TYPE "UDT_Recipe"
STRUCT
    name     : String[16];
    tempSet  : Real;
    mixTime  : Time;
END_STRUCT
END_TYPE
